FUNCTION_BLOCK FB_Manager
VAR
    arrLamper : ARRAY[1..10] OF POINTER TO FB_Lampe;
    iCount    : INT := 0;
END_VAR

METHOD Register
VAR_INPUT
    pLampe : POINTER TO FB_Lampe;
END_VAR
IF iCount < 10 THEN
    iCount := iCount + 1;
    arrLamper[iCount] := pLampe;
END_IF
END_METHOD

METHOD SlukAlle
VAR
    i : INT;
END_VAR
FOR i := 1 TO iCount DO
    arrLamper[i]^.bOn := FALSE;
END_FOR
END_METHOD

END_FUNCTION_BLOCK

(* stored: Version 1.1.0.1
   POU FB_Manager: Id {398e2c49-d1e7-4f1a-a149-f2a637033df5}, SpecialFunc None
   Method Register: Id {15aefec3-c231-4718-8dcc-dbc8b81c352a}
   Method SlukAlle: Id {3efb883d-f8f3-49bb-9437-e701be26ec8d} *)
